{attribute 'strict'}
{attribute 'to_string'}
TYPE eResult :
(
	NONE := 0,
	SUCCESS := 1,
	FAILURE := 2,
	ERROR	:= 3
);
END_TYPE

(* stored: Version 1.1.0.1, ProductVersion 3.1.4026.18
   DUT eResult: Id {99f9b0eb-e3b6-422c-9596-cf3bbef50d17} *)
